PROGRAM PRG_UpdatePhControl
VAR
	evtPhControlStart		: DetectEvent;
	evtPhControlStop		: DetectEvent;
	
END_VAR

evtPhControlStart(newSignalValue := phStart);
evtPhControlStop(newSignalValue := phStop);

IF evtPhControlStart.eventDetected = TASTEVT_PositiveEdge THEN
	phRunning := TRUE;
END_IF

IF evtPhControlStop.eventDetected = TASTEVT_PositiveEdge THEN
	phRunning := FALSE;
END_IF

IF pressureBar < 0.5 AND pressureBar > 0 AND phPumpManual THEN
	acidPumpSpeedCount := REAL_TO_INT(INT_TO_REAL(acidPumpSpeedSetting)*acidPumpSpeedCalibration.scaleFactor + acidPumpSpeedCalibration.offset);
	phPumpRunning := TRUE;
ELSE
	acidPumpSpeedCount := 0;
	phPumpRunning := FALSE;
END_IF

END_PROGRAM

(* stored: Version 1.1.0.1, ProductVersion 3.1.4022.7
   POU PRG_UpdatePhControl: Id {f1fc1e97-b3b8-412a-b5d4-e5b43139c85c}, SpecialFunc None *)
